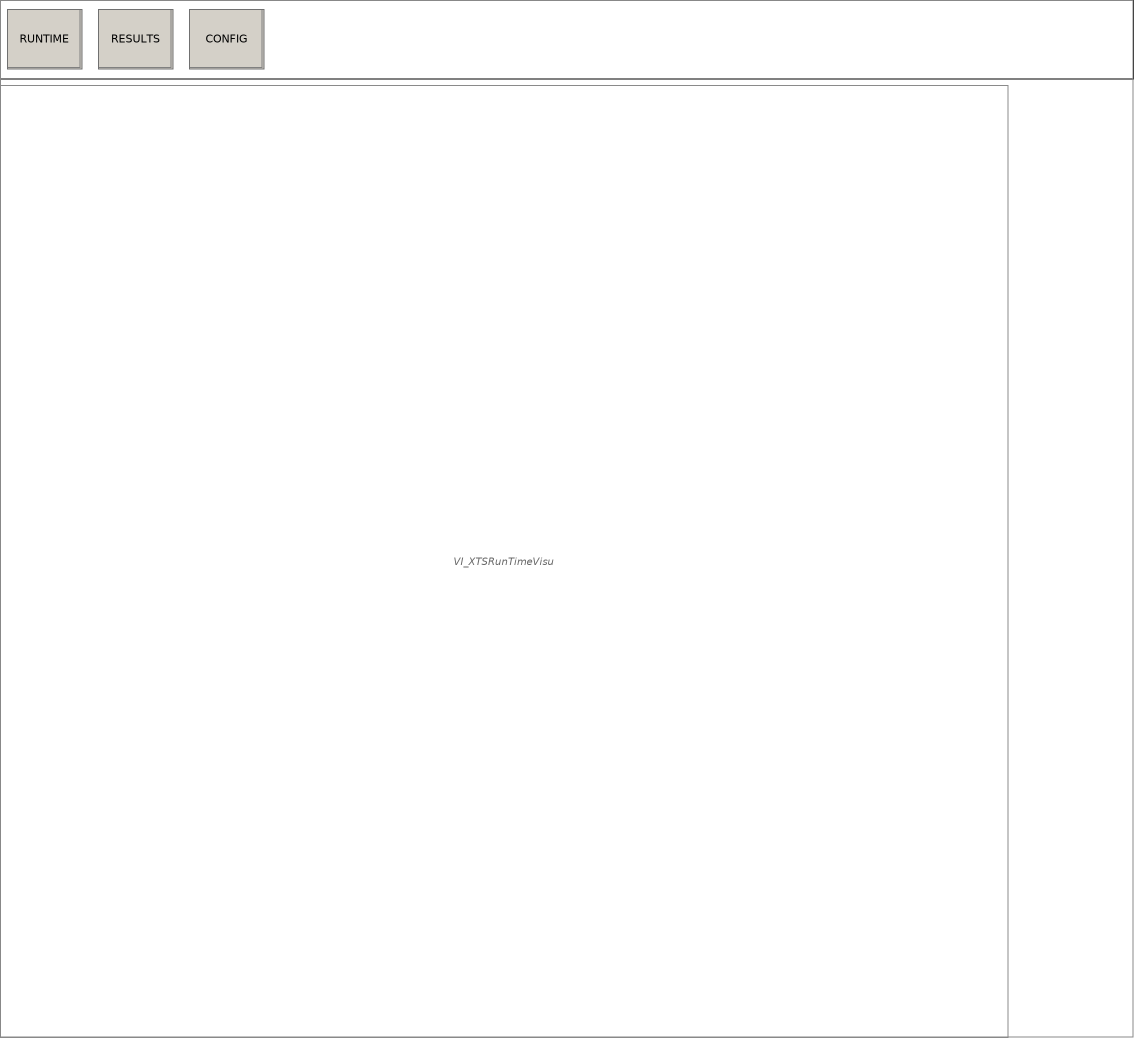
VISUALIZATION VI_XTSMainVisu  // 1134x1038
VAR_IN_OUT
	xts : XTS_System;
END_VAR
    Rectangle (0,0 1134x79)
    Button (7,9 75x60), "RUNTIME", colour toggle: xts.iFrameSelection=0
        OnMouseClick: execute { xts.iFrameSelection := 0; }
    Button (98,9 75x60), "RESULTS", colour toggle: xts.iFrameSelection=3
        OnMouseClick: execute { xts.iFrameSelection := 3; }
    Frame (0,85 1008x953), frame switch variable: xts.iFrameSelection
        shows VI_XTSRunTimeVisu(xts := xts)
        shows VI_XTSConfigurationVisu(xts := xts)
        shows VI_XTSMoversVisu(xts := xts)
        shows VI_XTSConfigurationVisu(xts := xts)
        shows VI_XTSManualVisu(xts := xts)
    Button (189,9 75x60), "CONFIG", colour toggle: xts.iFrameSelection=1
        OnMouseClick: execute { xts.iFrameSelection := 1; }
END_VISUALIZATION

(* stored: Version 1.1.0.1, ProductVersion 3.1.4024.11
   Visu VI_XTSMainVisu: Id {c4a25e79-daea-4b2a-873a-8fb188555ffe} *)
